TYPE ST_DeviceAddress :
STRUCT
	arrNetID		: ARRAY[0..5] OF BYTE;
	nPortNo			: UINT;
END_STRUCT
END_TYPE

(* stored: Version 1.1.0.1, ProductVersion 3.1.4024.15
   DUT ST_DeviceAddress: Id {5e5cfa2c-134f-4865-bfb2-e00108651ec6} *)
